PROGRAM MAIN
VAR
END_VAR

FOR hold := 1 TO 4 DO
	aLIghts[hold] := FALSE;
END_FOR

CASE CAS OF	
	0, 5..8:
	
		IF (NUM > 0) AND (NUM < 100) THEN;
			alights[1] := TRUE;
		
		ELSIF (NUM > 101) AND (NUM < 200) THEN;
			alights[2] := TRUE;
		END_IF
		
	1,2,3,4:
	
		IF (NUM > 201) AND (NUM < 300) THEN;
			alights[3] := TRUE;
		
		ELSIF (NUM > 301) AND (NUM < 400) THEN;
			alights[4] := TRUE;
			
		END_IF	
	
END_CASE
	
IF test := TRUE THEN;
	robo1.aDirection[1] := TRUE;
	
	robo2.aDirection[3] := TRUE;
END_IF


POU();

END_PROGRAM

(* stored: Version 1.1.0.1, ProductVersion 3.1.4024.12
   POU MAIN: Id {e9c7b7b8-0d44-4f84-a605-4e636016ba56}, SpecialFunc None *)
